TYPE ST_ENCODER_OUT :
STRUCT
	bDeviceDisable			: BOOL;

	nRevolutions			: UDINT := 0;
	nPulses				: UDINT;
	fPositionInMM			: LREAL;

	bError					: BOOL;
	sError					: STRING;

	nWarningStatus		: UINT;
	nAlarmStatus			: UINT;

END_STRUCT
END_TYPE

(* stored: Version 1.1.0.1
   DUT ST_ENCODER_OUT: Id {fe17c430-3140-454c-87c9-5ee52f941489} *)
